TYPE ST_RejectReasonOUT3 :
STRUCT
	Reason	:STRING;
END_STRUCT
END_TYPE

(* stored: Version 1.1.0.1, ProductVersion 3.1.4024.13
   DUT ST_RejectReasonOUT3: Id {87c704d0-614c-4a4e-98ab-b69c72cc1fad} *)
